// Mitsubishi GX Works2 project: pulse1   PLC: Q03UDV

PROGRAM MAIN
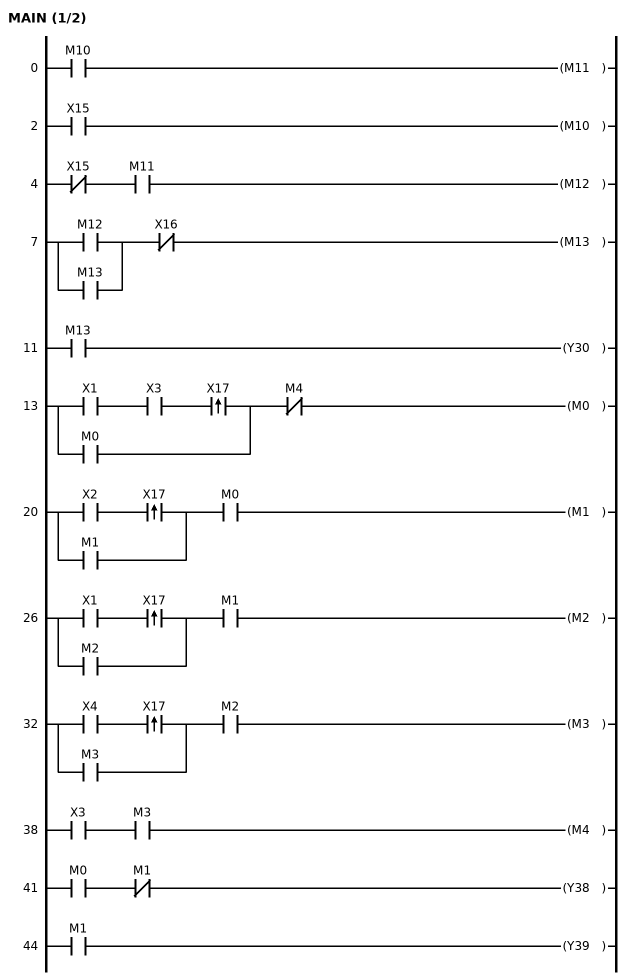
0     LD      M10
      OUT     M11
2     LD      X15
      OUT     M10
4     LDI     X15
      AND     M11
      OUT     M12
7     LD      M12
      OR      M13
      ANI     X16
      OUT     M13
11    LD      M13
      OUT     Y30
13    LD      X1
      AND     X3
      ANDP    X17
      OR      M0
      ANI     M4
      OUT     M0
20    LD      X2
      ANDP    X17
      OR      M1
      AND     M0
      OUT     M1
26    LD      X1
      ANDP    X17
      OR      M2
      AND     M1
      OUT     M2
32    LD      X4
      ANDP    X17
      OR      M3
      AND     M2
      OUT     M3
38    LD      X3
      AND     M3
      OUT     M4
41    LD      M0
      ANI     M1
      OUT     Y38
44    LD      M1
      OUT     Y39
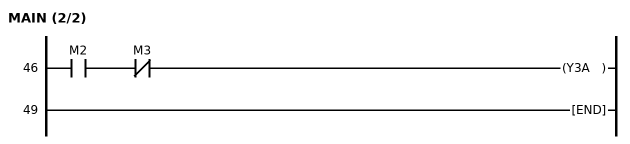
46    LD      M2
      ANI     M3
      OUT     Y3A
49    END
END_PROGRAM
